FUNCTION_BLOCK AandCReactants (* Composite Function Block Type *)
  (* Standard: 61499-2 *)
  (* Version 0.0, 2018-10-14, 4DIAC-IDE, 4DIAC-Consortium *)
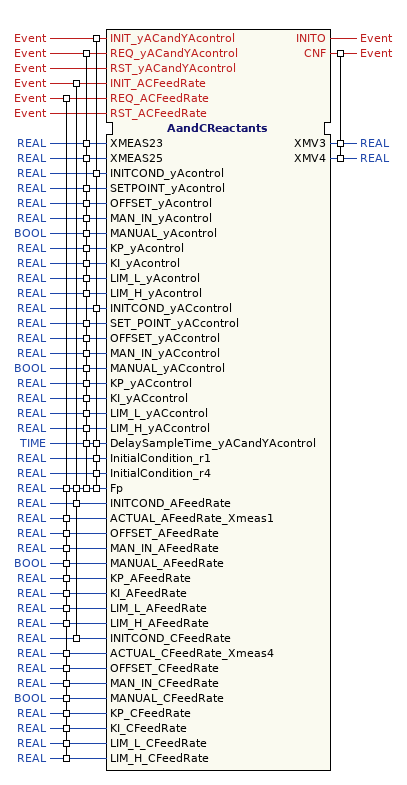
  EVENT_INPUT
    INIT_yACandYAcontrol WITH INITCOND_yAcontrol, INITCOND_yACcontrol, DelaySampleTime_yACandYAcontrol, InitialCondition_r1, InitialCondition_r4, Fp; (* Initialization Request *)
    REQ_yACandYAcontrol WITH XMEAS23, XMEAS25, SETPOINT_yAcontrol, OFFSET_yAcontrol, MAN_IN_yAcontrol, MANUAL_yAcontrol, LIM_L_yAcontrol, KP_yAcontrol, KI_yAcontrol, LIM_H_yAcontrol, SET_POINT_yACcontrol, OFFSET_yACcontrol, MAN_IN_yACcontrol, MANUAL_yACcontrol, DelaySampleTime_yACandYAcontrol, LIM_H_yACcontrol, LIM_L_yACcontrol, KI_yACcontrol, KP_yACcontrol, Fp; (* Normal Execution Request *)
    RST_yACandYAcontrol;
    INIT_ACFeedRate WITH Fp, INITCOND_AFeedRate, INITCOND_CFeedRate;
    REQ_ACFeedRate WITH Fp, ACTUAL_AFeedRate_Xmeas1, OFFSET_AFeedRate, MAN_IN_AFeedRate, MANUAL_AFeedRate, KP_AFeedRate, KI_AFeedRate, LIM_L_AFeedRate, LIM_H_AFeedRate, ACTUAL_CFeedRate_Xmeas4, OFFSET_CFeedRate, MAN_IN_CFeedRate, MANUAL_CFeedRate, KP_CFeedRate, KI_CFeedRate, LIM_L_CFeedRate, LIM_H_CFeedRate;
    RST_ACFeedRate;
  END_EVENT
  EVENT_OUTPUT
    INITO; (* Initialization Confirm *)
    CNF WITH XMV3, XMV4; (* Execution Confirmation *)
  END_EVENT
  VAR_INPUT
    XMEAS23 : REAL;
    XMEAS25 : REAL;
    INITCOND_yAcontrol : REAL;
    SETPOINT_yAcontrol : REAL;
    OFFSET_yAcontrol : REAL;
    MAN_IN_yAcontrol : REAL;
    MANUAL_yAcontrol : BOOL;
    KP_yAcontrol : REAL;
    KI_yAcontrol : REAL;
    LIM_L_yAcontrol : REAL;
    LIM_H_yAcontrol : REAL;
    INITCOND_yACcontrol : REAL;
    SET_POINT_yACcontrol : REAL;
    OFFSET_yACcontrol : REAL;
    MAN_IN_yACcontrol : REAL;
    MANUAL_yACcontrol : BOOL;
    KP_yACcontrol : REAL;
    KI_yACcontrol : REAL;
    LIM_L_yACcontrol : REAL;
    LIM_H_yACcontrol : REAL;
    DelaySampleTime_yACandYAcontrol : TIME;
    InitialCondition_r1 : REAL;
    InitialCondition_r4 : REAL;
    Fp : REAL;
    INITCOND_AFeedRate : REAL;
    ACTUAL_AFeedRate_Xmeas1 : REAL;
    OFFSET_AFeedRate : REAL;
    MAN_IN_AFeedRate : REAL;
    MANUAL_AFeedRate : BOOL;
    KP_AFeedRate : REAL;
    KI_AFeedRate : REAL;
    LIM_L_AFeedRate : REAL;
    LIM_H_AFeedRate : REAL;
    INITCOND_CFeedRate : REAL;
    ACTUAL_CFeedRate_Xmeas4 : REAL;
    OFFSET_CFeedRate : REAL;
    MAN_IN_CFeedRate : REAL;
    MANUAL_CFeedRate : BOOL;
    KP_CFeedRate : REAL;
    KI_CFeedRate : REAL;
    LIM_L_CFeedRate : REAL;
    LIM_H_CFeedRate : REAL;
  END_VAR
  VAR_OUTPUT
    XMV3 : REAL;
    XMV4 : REAL;
  END_VAR
  FBS
    REAL2REAL : REAL2REAL(IN := 100);
    F_MUL : F_MUL;
    xmeas23x100 : REAL2REAL;
    yA : F_DIV;
    F_ADD : F_ADD;
    yAC : REAL2REAL;
    yAcontrol : FB_CTRL_PI;
    yACcontrol : FB_CTRL_PI;
    loo14 : F_ADD;
    Delayr1 : Delay_With_InitConditionREALtype;
    r1 : REAL2REAL;
    Fpxr1 : F_MUL;
    AFeedRate : FB_CTRL_PI;
    InitXMV3 : Init_ConditionREALtype;
    F_SUB : F_SUB;
    loop15minloop14 : REAL2REAL;
    r4_ : F_ADD;
    delayr4 : Delay_With_InitConditionREALtype;
    F_MUL_1 : F_MUL;
    REAL2REAL_1 : REAL2REAL;
    CFeedRate : FB_CTRL_PI;
    InitXMV4 : Init_ConditionREALtype;
    Init_ConditionREALtype : Init_ConditionREALtype;
    Init_ConditionREALtype_1 : Init_ConditionREALtype;
  END_FBS
  EVENT_CONNECTIONS
    REQ_yACandYAcontrol TO REAL2REAL.REQ;
    REAL2REAL.CNF TO F_MUL.REQ;
    F_MUL.CNF TO xmeas23x100.REQ;
    xmeas23x100.CNF TO yA.REQ;
    REQ_yACandYAcontrol TO F_ADD.REQ;
    INIT_yACandYAcontrol TO INITO;
    F_ADD.CNF TO yAC.REQ;
    yAC.CNF TO yA.REQ;
    yA.CNF TO yAcontrol.REQ;
    INIT_yACandYAcontrol TO yAcontrol.INIT;
    yAcontrol.INITO TO yACcontrol.INIT;
    yAC.CNF TO yACcontrol.REQ;
    REQ_yACandYAcontrol TO yACcontrol.REQ;
    REQ_yACandYAcontrol TO yAcontrol.REQ;
    loo14.CNF TO Delayr1.Start_and_REQ;
    yAcontrol.INITO TO Delayr1.INIT;
    Delayr1.CNF TO loo14.REQ;
    loo14.CNF TO r1.REQ;
    r1.CNF TO Fpxr1.REQ;
    AFeedRate.INITO TO InitXMV3.InitEvent;
    AFeedRate.CNF TO InitXMV3.SubsequentEvent;
    F_SUB.CNF TO loop15minloop14.REQ;
    loop15minloop14.CNF TO r4_.REQ;
    yACcontrol.INITO TO delayr4.INIT;
    r4_.CNF TO delayr4.Start_and_REQ;
    delayr4.CNF TO r4_.REQ;
    r4_.CNF TO REAL2REAL_1.REQ;
    REAL2REAL_1.CNF TO F_MUL_1.REQ;
    CFeedRate.INITO TO InitXMV4.InitEvent;
    CFeedRate.CNF TO InitXMV4.SubsequentEvent;
    RST_yACandYAcontrol TO yAcontrol.RST;
    RST_yACandYAcontrol TO yACcontrol.RST;
    yAcontrol.INITO TO Init_ConditionREALtype.InitEvent;
    yAcontrol.CNF TO Init_ConditionREALtype.SubsequentEvent;
    Init_ConditionREALtype.CNF TO loo14.REQ;
    yACcontrol.INITO TO Init_ConditionREALtype_1.InitEvent;
    Init_ConditionREALtype.CNF TO F_SUB.REQ;
    yACcontrol.CNF TO Init_ConditionREALtype_1.SubsequentEvent;
    Init_ConditionREALtype_1.CNF TO F_SUB.REQ;
    InitXMV4.CNF TO CNF;
    InitXMV3.CNF TO CNF;
    Fpxr1.CNF TO AFeedRate.REQ;
    INIT_ACFeedRate TO AFeedRate.INIT;
    REQ_ACFeedRate TO AFeedRate.REQ;
    RST_ACFeedRate TO AFeedRate.RST;
    INIT_ACFeedRate TO CFeedRate.INIT;
    REQ_ACFeedRate TO CFeedRate.REQ;
    RST_ACFeedRate TO CFeedRate.RST;
    F_MUL_1.CNF TO CFeedRate.REQ;
    REQ_ACFeedRate TO F_MUL_1.REQ;
    REQ_ACFeedRate TO Fpxr1.REQ;
    AFeedRate.INITO TO INITO;
    CFeedRate.INITO TO INITO;
  END_CONNECTIONS
  DATA_CONNECTIONS
    REAL2REAL.OUT TO F_MUL.IN2;
    XMEAS23 TO F_MUL.IN1;
    F_MUL.OUT TO xmeas23x100.IN;
    xmeas23x100.OUT TO yA.IN1;
    XMEAS23 TO F_ADD.IN1;
    XMEAS25 TO F_ADD.IN2;
    F_ADD.OUT TO yAC.IN;
    yAC.OUT TO yA.IN2;
    yA.OUT TO yAcontrol.ACTUAL;
    SETPOINT_yAcontrol TO yAcontrol.SET_POINT;
    OFFSET_yAcontrol TO yAcontrol.OFFSET;
    MAN_IN_yAcontrol TO yAcontrol.MAN_IN;
    MANUAL_yAcontrol TO yAcontrol.MANUAL;
    KP_yAcontrol TO yAcontrol.KP;
    KI_yAcontrol TO yAcontrol.KI;
    LIM_L_yAcontrol TO yAcontrol.LIM_L;
    LIM_H_yAcontrol TO yAcontrol.LIM_H;
    yAC.OUT TO yACcontrol.ACTUAL;
    SET_POINT_yACcontrol TO yACcontrol.SET_POINT;
    OFFSET_yACcontrol TO yACcontrol.OFFSET;
    MAN_IN_yACcontrol TO yACcontrol.MAN_IN;
    MANUAL_yACcontrol TO yACcontrol.MANUAL;
    KP_yACcontrol TO yACcontrol.KP;
    KI_yACcontrol TO yACcontrol.KI;
    LIM_L_yACcontrol TO yACcontrol.LIM_L;
    LIM_H_yACcontrol TO yACcontrol.LIM_H;
    DelaySampleTime_yACandYAcontrol TO Delayr1.DelayTime;
    InitialCondition_r1 TO Delayr1.InitialCondition;
    loo14.OUT TO Delayr1.DelayedInput;
    Delayr1.OUT TO loo14.IN2;
    loo14.OUT TO r1.IN;
    r1.OUT TO Fpxr1.IN1;
    Fp TO Fpxr1.IN2;
    Fpxr1.OUT TO AFeedRate.SET_POINT;
    AFeedRate.Y TO InitXMV3.SubsequentInput;
    INITCOND_AFeedRate TO InitXMV3.InitialCondition;
    ACTUAL_AFeedRate_Xmeas1 TO AFeedRate.ACTUAL;
    OFFSET_AFeedRate TO AFeedRate.OFFSET;
    MAN_IN_AFeedRate TO AFeedRate.MAN_IN;
    MANUAL_AFeedRate TO AFeedRate.MANUAL;
    KP_AFeedRate TO AFeedRate.KP;
    KI_AFeedRate TO AFeedRate.KI;
    LIM_L_AFeedRate TO AFeedRate.LIM_L;
    LIM_H_AFeedRate TO AFeedRate.LIM_H;
    F_SUB.OUT TO loop15minloop14.IN;
    loop15minloop14.OUT TO r4_.IN1;
    r4_.OUT TO delayr4.DelayedInput;
    DelaySampleTime_yACandYAcontrol TO delayr4.DelayTime;
    InitialCondition_r4 TO delayr4.InitialCondition;
    delayr4.OUT TO r4_.IN2;
    r4_.OUT TO REAL2REAL_1.IN;
    REAL2REAL_1.OUT TO F_MUL_1.IN1;
    Fp TO F_MUL_1.IN2;
    F_MUL_1.OUT TO CFeedRate.SET_POINT;
    CFeedRate.Y TO InitXMV4.SubsequentInput;
    INITCOND_CFeedRate TO InitXMV4.InitialCondition;
    ACTUAL_CFeedRate_Xmeas4 TO CFeedRate.ACTUAL;
    OFFSET_CFeedRate TO CFeedRate.OFFSET;
    MAN_IN_CFeedRate TO CFeedRate.MAN_IN;
    MANUAL_CFeedRate TO CFeedRate.MANUAL;
    KP_CFeedRate TO CFeedRate.KP;
    KI_CFeedRate TO CFeedRate.KI;
    LIM_L_CFeedRate TO CFeedRate.LIM_L;
    LIM_H_CFeedRate TO CFeedRate.LIM_H;
    yAcontrol.Y TO Init_ConditionREALtype.SubsequentInput;
    Init_ConditionREALtype.OUT TO loo14.IN1;
    Init_ConditionREALtype.OUT TO F_SUB.IN2;
    Init_ConditionREALtype_1.OUT TO F_SUB.IN1;
    yACcontrol.Y TO Init_ConditionREALtype_1.SubsequentInput;
    INITCOND_yAcontrol TO Init_ConditionREALtype.InitialCondition;
    INITCOND_yACcontrol TO Init_ConditionREALtype_1.InitialCondition;
    InitXMV3.OUT TO XMV3;
    InitXMV4.OUT TO XMV4;
  END_CONNECTIONS
END_FUNCTION_BLOCK
